(* IEC 61131-3 sources: volt/packages/volt-lsp-iec/test-corpus/lenze-mid/Device/Plc Logic/Application/Library Manager/(unresolved)/cmpeventmgr interfaces, 5 files *)

(* ---- EVENTPARAM.dut ---- *)
TYPE EVENTPARAM :
STRUCT
	EVENTID : DWORD;
	CMPIDPROVIDER : DWORD;
	USPARAMID : WORD;
	USVERSION : WORD;
	PPARAMETER : POINTER TO BYTE;
END_STRUCT
END_TYPE

(* ---- EVENTPARAM2.dut ---- *)
TYPE EVENTPARAM2 :
STRUCT
	EVENTID : DWORD;
	CMPIDPROVIDER : DWORD;
	USPARAMID : WORD;
	USVERSION : WORD;
	PPARAMETER : POINTER TO BYTE;
	PUSERPARAMETER : POINTER TO BYTE;
END_STRUCT
END_TYPE

(* ---- CONSTANTS.gvl ---- *)
VAR_GLOBAL
	EVENT_CALLBACKS_NO_LIMIT : UDINT := 16#FFFFFFFF;
	CMPID_CMPEVENTMGR : UDINT := 16#5B;
	ITFID_ICMPEVENTCALLBACK : UDINT := 16#25;
END_VAR

(* ---- EVENTCLASS.gvl ---- *)
VAR_GLOBAL
	EVTCLASS_NONE : UINT := 0;
	EVTCLASS_ALL : UINT := 16#FFFF;
	EVTCLASS_INFO : UINT := 16#1;
	EVTCLASS_WARNING : UINT := 16#2;
	EVTCLASS_ERROR : UINT := 16#4;
	EVTCLASS_EXCEPTION : UINT := 16#8;
	EVTCLASS_VENDOR_SPEC : UINT := 16#1000;
END_VAR

(* ---- ICMPEVENTCALLBACK.itf ---- *)
INTERFACE ICMPEVENTCALLBACK
END_INTERFACE

METHOD EVENTCALLBACK : RTS_IEC_RESULT
VAR_INPUT
	PEVENTPARAM : POINTER TO EventParam;
END_VAR
END_METHOD
